(*P&ID: 2 cylinder but Actual design 1 cylinder1*)
FUNCTION_BLOCK FB_TankFill_2Cylinder IMPLEMENTS I_TankFill
VAR
	poCylinder1 : FB_DigitalOutput;
	poCylinder2 : FB_DigitalOutput;
END_VAR

poCylinder1();
poCylinder2();

METHOD Close : BOOL
VAR_INPUT
END_VAR
poCylinder1.Out := FALSE;
poCylinder2.Out := FALSE;
END_METHOD

PROPERTY IsClose : bool
GET
IsClose := poCylinder1.Out=false;
END_GET
END_PROPERTY

PROPERTY IsOpen : bool
GET
IsOpen := poCylinder1.Out=True;
END_GET
END_PROPERTY

METHOD Open : BOOL
VAR_INPUT
END_VAR
poCylinder1.Out := TRUE;
poCylinder2.Out := TRUE;
END_METHOD

PROPERTY Ref_poCylinder1 : Reference to FB_DigitalOutput
GET
Ref_poCylinder1 ref= poCylinder1;
END_GET
END_PROPERTY

PROPERTY Ref_poCylinder2 : Reference to FB_DigitalOutput
GET
Ref_poCylinder2 ref= poCylinder2;
END_GET
END_PROPERTY

END_FUNCTION_BLOCK

(* stored: Version 1.1.0.1, ProductVersion 3.1.4024.12
   POU FB_TankFill_2Cylinder: Id {e8944d61-9ce1-41f9-874d-840296d361ce}, SpecialFunc None
   Method Close: Id {afd8bf84-8924-40d9-9ece-bcd22d73ad2b}
   Property IsClose: Id {b2b0c821-38ac-4afd-9f9c-9e4c85d09fb8}
   Get Get: Id {90616937-43c3-4663-abf8-b01c76fe1d28}
   Property IsOpen: Id {f2fd2810-e07e-42b2-853a-ddd42eab6f36}
   Get Get: Id {647f5201-07e6-4ee0-90b4-f5d3816af186}
   Method Open: Id {bdd526e2-4452-4c08-a6cf-31733794465b}
   Property Ref_poCylinder1: Id {a5b7aee3-8e80-4a76-95be-4212e4e33b4f}
   Get Get: Id {b2ed88a1-6839-4a02-bcc9-c62bc55f3227}
   Property Ref_poCylinder2: Id {ff372483-ae3c-4298-a684-803846f48b11}
   Get Get: Id {33410d3b-27b2-4809-a684-c7784cb9bc0b} *)
